Universal Robots PolyScope program: vision.urp

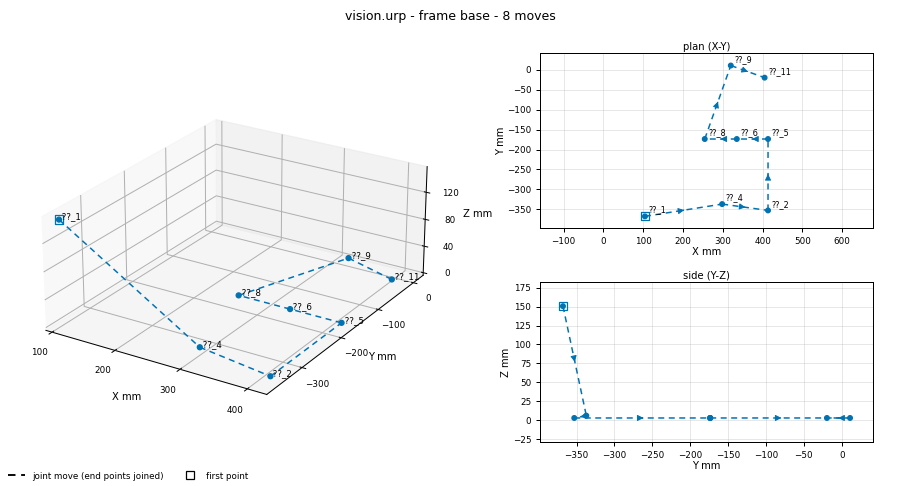
[picture p0: tool path of vision.urp in frame base, 8 of 16 moves have a stored position in this frame; points joined in program order, loops and branches not executed]
Program vision (installation=20240827 directory=/programs/show createdIn=5.13.1 lastSavedIn=5.15.1 robotSerialNumber=20245500285)
Calibrated DH parameters: a=[0.000097, -0.210459, -0.026602, 0.000137, 0.000078, 0]; d=[0.162601, 254.180657, -54.076236, -199.970743, 0.099615, 0.099684]; alpha=[1.569796, -0.001455, 0.001957, 1.570525, -1.571561, 0]; deltaTheta=[0, -1.053331, 8.839472, -1.50296, 0.000002, 0]
InitVariablesNode
Robot Program (runOnlyOnce=false)
  'set tcp'
  If False
    'begin'
    MoveJ speed 180 deg/s, acceleration 400 deg/s^2 (useActiveTCP=true positionType=JointAngles) feature=Base
      Waypoint 路点_1: TCP in base x=104.511 y=-367.887 z=150.56 mm, rx=-1.9493 ry=-1.8262 rz=-0.6048 rad; joints [85.471, -80.224, 100.082, -75.625, -90.165, 89.439] deg; TCP offset x=-0.17 y=0 z=192.95 mm, rx=0 ry=0 rz=0 rad
    'target'
    MoveJ speed 180 deg/s, acceleration 400 deg/s^2 (useActiveTCP=true) feature=Base
      Waypoint 路点_4: TCP in base x=298.358 y=-337.063 z=6.061 mm, rx=2.219 ry=2.2146 rz=-0.0019 rad; joints [114.12, -81.962, 128.733, -137.191, -90, 114.383] deg
      Waypoint 路点_2: TCP in base x=413.589 y=-352.997 z=2.997 mm, rx=2.2212 ry=2.221 rz=0.0029 rad; joints [125.153, -70.625, 113.787, -133.215, -89.966, 125.322] deg
      Waypoint 路点_5: TCP in base x=413.621 y=-173.641 z=3 mm, rx=2.221 ry=2.2212 rz=0.0029 rad; joints [139.755, -81.637, 128.862, -137.305, -89.965, 139.9] deg; TCP offset x=-0.17 y=0 z=192.95 mm, rx=0 ry=0 rz=0 rad
      Waypoint 路点_6: TCP in base x=335.16 y=-173.643 z=3 mm, rx=2.2211 ry=2.2211 rz=0.0029 rad; joints [131.722, -91.143, 139.321, -138.241, -89.956, 131.857] deg; TCP offset x=-0.17 y=0 z=192.95 mm, rx=0 ry=0 rz=0 rad
      Waypoint 路点_8: TCP in base x=254.659 y=-173.63 z=3 mm, rx=2.2212 ry=2.2211 rz=0.0029 rad; joints [119.834, -102.953, 148.816, -135.903, -89.943, 119.958] deg; TCP offset x=-0.17 y=0 z=192.95 mm, rx=0 ry=0 rz=0 rad
      Waypoint 路点_9: TCP in base x=320.034 y=10.925 z=3.003 mm, rx=2.2211 ry=2.2212 rz=0.0029 rad; joints [157.143, -100.627, 147.26, -136.739, -89.964, 157.268] deg; TCP offset x=-0.17 y=0 z=192.95 mm, rx=0 ry=0 rz=0 rad
      Waypoint 路点_11: TCP in base x=405.002 y=-19.56 z=2.994 mm, rx=2.2212 ry=2.2211 rz=0.0029 rad; joints [157.861, -87.192, 135.295, -138.21, -89.977, 158.004] deg
  '########'
  'set var'
  begin_pos := 路点_1
  h_up := 0.1
  var_1 := 路点_2
  var_2 := 路点_4
  var_3 := 路点_5
  var_4 := 路点_6
  var_5 := 路点_8
  var_6 := 路点_11
  var_7 := 路点_9
  tcp := [var_1,var_2,var_3,var_4,var_5,var_6,var_7]
  '##########'
  'run'
  MoveJ speed 180 deg/s, acceleration 400 deg/s^2 (useActiveTCP=true positionType=JointAngles) feature=Base
    Waypoint Variable (Variable): variable(name=begin_pos)
  Script: vision = rpc_factory("xmlrpc","http://192.168.1.7:9121/RPC2")
  Script: gripper = rpc_factory("xmlrpc","http://192.168.1.7:9120/RPC2")
  Script: gripper.open()
  Loop Forever
    n := 0
    MoveJ speed 180 deg/s, acceleration 400 deg/s^2 (useActiveTCP=true positionType=JointAngles) feature=Base
      Waypoint Variable (Variable): variable=begin_pos
    Popup Message (haltProgram=false message=photo inputType=Text)
    campose := get_actual_tcp_pose()
    take := True
    Loop While (checkContinuously=false) expression=take== True
      photo := vision.take_photo(campose)
      If photo≠ True
        Popup Message (haltProgram=false message=continues? inputType=Text)
      Else 
        take := False
    articlenum := vision.get_obj_num()
    SuppressedNode
      Popup Message (haltProgram=false message=articlenum inputType=Variable) variable=articlenum
    SuppressedNode
      mode := 0
    If articlenum>7
      Popup Warning (haltProgram=false message=over max obj inputType=Text)
      SuppressedNode
        mode := 1
    Loop While (checkContinuously=false) expression=n<articlenum
      obj_num := n
      pose := p[0.0,0.0,0.0,2.221,2.221,0.004]
      obj_pose := vision.get_obj_pose(obj_num)
      Script: pose[0]=obj_pose[0]
      Script: pose[1]=obj_pose[1]
      Script: pose[2]=obj_pose[2]+0.025
      Script: pose[3]=obj_pose[3]
      Script: pose[4]=obj_pose[4]
      Script: pose[5]=obj_pose[5]
      MoveL speed 3000 mm/s, acceleration 6000 mm/s^2 (useActiveTCP=true) feature=Base
        Waypoint Variable (Variable): variable(name=pose)
      Script: pose[2]=obj_pose[2] - 0.06
      If pose[2]<0.003
        Script: pose[2] = 0.003
      MoveL speed 3000 mm/s, acceleration 6000 mm/s^2 (useActiveTCP=true) feature=Base
        Waypoint Variable (Variable): variable=pose
        Script: gripper.adaptiveClose()
      first_pose := pose
      Script: pose[2]=pose[2] + h_up
      MoveL speed 3000 mm/s, acceleration 6000 mm/s^2 (useActiveTCP=true) feature=Base
        Waypoint Variable (Variable): variable=pose
      target_pose := tcp[n]
      Script: target_pose[2]=first_pose[2]
      down_pose := target_pose
      Script: down_pose[2]=down_pose[2] + h_up
      MoveL speed 3000 mm/s, acceleration 6000 mm/s^2 (useActiveTCP=true) feature=Base
        Waypoint Variable (Variable): variable(name=down_pose)
      MoveL speed 3000 mm/s, acceleration 6000 mm/s^2 (useActiveTCP=true) feature=Base
        Waypoint Variable (Variable): variable(name=target_pose)
        Script: gripper.open()
      MoveL speed 3000 mm/s, acceleration 6000 mm/s^2 (useActiveTCP=true) feature=Base
        Waypoint Variable (Variable): variable=down_pose
      n := n + 1
  '########################'
